FUNCTION_BLOCK Model (* Composite Function Block Type *)
  (* Standard: 61499-2 *)
  (* Version 0.0, 6/17/2016, Andrei, nxtControl GmbH, template *)
  PACKAGE Main;
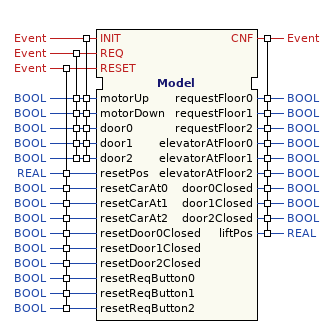
  EVENT_INPUT
    INIT WITH motorUp, motorDown, door0, door1, door2; (* Initialization Request *)
    REQ WITH motorUp, motorDown, door0, door1, door2; (* Normal Execution Request *)
    RESET WITH resetPos, resetCarAt0, resetCarAt1, resetCarAt2, resetDoor0Closed, resetDoor1Closed, resetDoor2Closed, resetReqButton0, resetReqButton1, resetReqButton2;
  END_EVENT
  EVENT_OUTPUT
    CNF WITH requestFloor0, requestFloor1, requestFloor2, elevatorAtFloor0, elevatorAtFloor1, elevatorAtFloor2, door0Closed, door1Closed, door2Closed, liftPos; (* Execution Confirmation *)
  END_EVENT
  VAR_INPUT
    motorUp : BOOL; (* Input event qualifier *)
    motorDown : BOOL;
    door0 : BOOL;
    door1 : BOOL;
    door2 : BOOL;
    resetPos : REAL;
    resetCarAt0 : BOOL;
    resetCarAt1 : BOOL;
    resetCarAt2 : BOOL;
    resetDoor0Closed : BOOL;
    resetDoor1Closed : BOOL;
    resetDoor2Closed : BOOL;
    resetReqButton0 : BOOL;
    resetReqButton1 : BOOL;
    resetReqButton2 : BOOL;
  END_VAR
  VAR_OUTPUT
    requestFloor0 : BOOL;
    requestFloor1 : BOOL;
    requestFloor2 : BOOL;
    elevatorAtFloor0 : BOOL;
    elevatorAtFloor1 : BOOL;
    elevatorAtFloor2 : BOOL;
    door0Closed : BOOL;
    door1Closed : BOOL;
    door2Closed : BOOL;
    liftPos : REAL; (* Output event qualifier *)
  END_VAR
  FBS
    FB1 : Lift;
    Doors : Doors;
    FB3 : ReqPanelLift;
    FB4 : FloorCarElevator;
  END_FBS
  EVENT_CONNECTIONS
    REQ TO FB1.REQ;
    INIT TO FB1.INIT;
    FB1.CNF TO FB4.REQ;
    FB4.CNF TO Doors.REQ;
    FB1.INITO TO Doors.INIT;
    FB3.CNF TO CNF;
    FB3.INITO TO FB1.REQ;
    RESET TO FB1.RESET;
    FB1.RESOUT TO FB4.RESET;
    FB4.RESOUT TO Doors.RESET;
    Doors.INITO TO FB3.INIT;
    Doors.CNF TO FB3.REQ;
    Doors.RESOUT TO FB3.RESET;
  END_CONNECTIONS
  DATA_CONNECTIONS
    motorUp TO FB1.MoveUp;
    motorDown TO FB1.MoveDown;
    FB3.ButtonFor0 TO requestFloor0;
    FB3.ButtonFor1 TO requestFloor1;
    FB3.ButtonFor2 TO requestFloor2;
    FB1.LiftPos TO FB4.CarPos;
    FB4.CarAt0 TO FB3.LiftAt0;
    FB4.CarAt1 TO FB3.LiftAt1;
    FB4.CarAt2 TO FB3.LiftAt2;
    FB4.CarAt2 TO elevatorAtFloor2;
    FB4.CarAt1 TO elevatorAtFloor1;
    FB4.CarAt0 TO elevatorAtFloor0;
    FB1.LiftPos TO liftPos;
    door1 TO Doors.door1Open;
    Doors.door0Closed TO door0Closed;
    Doors.door1Closed TO door1Closed;
    Doors.door2Closed TO door2Closed;
    door0 TO Doors.door0Open;
    resetPos TO FB1.resetPos;
    resetCarAt1 TO FB4.resetCarAt1;
    resetCarAt2 TO FB4.resetCarAt2;
    resetDoor0Closed TO Doors.resetDoor0Closed;
    resetDoor1Closed TO Doors.resetDoor1Closed;
    resetDoor2Closed TO Doors.resetDoor2Closed;
    resetReqButton0 TO FB3.ResetReqButton0;
    resetReqButton1 TO FB3.ResetReqButton1;
    resetReqButton2 TO FB3.ResetReqButton2;
    resetCarAt0 TO FB4.resetCarAt0;
    door2 TO Doors.door2Open;
    Doors.Door0Opened TO FB3.DoorOpen0;
    Doors.Door1Opened TO FB3.DoorOpen1;
    Doors.Door2Opened TO FB3.DoorOpen2;
  END_CONNECTIONS
END_FUNCTION_BLOCK
